KUKA KRL data list: user_sps.dat

&ACCESS RVP1
&REL 14
&COMMENT User SPS V1.0
DEFDAT  User_SPS PUBLIC
Global ENUM TSPS_MOD _Init,_Loop


ENDDAT
